(* Logix 5000 project; controller Drives_Line1 1756-L72 rev 20.13; software revision 20.04; part 11 of 21 *)
(* tags used below, declared in another part *)
   Bridle_02_FB_Count_Old : DINT;
   Bridle_02_Max_FBcounts : REAL;
   Bridle_02_SpdTrimMPS : REAL;
   Bridle_02_SpdTrimPct : REAL;
   Bridle_02a_RPMPerMPS : REAL;
   Bridle_02b_RPMPerMPS : REAL;
   IO_State_Bridle_02a : INT;
   IO_State_Bridle_02b : INT;
   IO_State_Tmp_Bridle_02a : INT;
   IO_State_Tmp_Bridle_02b : INT;
   Ons : DINT;
   PulsReset_PID : TIMER;
   TimeOn_PIDOn : TIMER;
   TofReset : TIMER;
   TonNoResponse : TIMER[3];
   TonRefOn : TIMER;
   zBridle_02_Ki_SpdTrim : REAL;
   zBridle_02_Kp_SpdTrim : REAL;
   zBridle_02_Max_rev : DINT;
   zBridle_02_MaxAccDec : REAL;
   zBridle_02_MaxTrimSpdTrim : REAL;
   zBridle_02_MinTrimSpdTrim : REAL;
   zBridle_02b_EncRes : DINT;
   Bridle_02 : UDT_Bridle_2M;
   Bridle_02_FB_Diff : DINT;
   Bridle_02_FB_Update_Valid : BOOL;
   Bridle_02_Rev_mm : REAL;
   Bridle_02b_FBCounts_mm : DINT;
   EntryCtrl : UDT_Control_Zone;
   In_Commands : UDT_Commands;
   In_Config : UDT_Config;
   LineCmd : UDT_Commands_Line;
   LineCtrl : UDT_Control_Line;
   LineFdbks : UDT_Feedbacks_Line;
   TaskInterval_ms : DINT;
   zConfigFromMaster : BOOL;
   zPi : REAL;
   zSimulation : BOOL;
(* P15_Bridle_02, continued *)

ROUTINE R01_From_Master   (* ladder *)
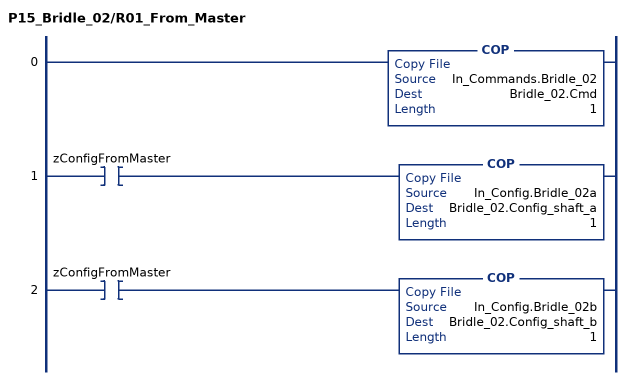
   0: COP(In_Commands.Bridle_02,Bridle_02.Cmd,1);
   1: XIC(zConfigFromMaster)COP(In_Config.Bridle_02a,Bridle_02.Config_shaft_a,1);
   2: XIC(zConfigFromMaster)COP(In_Config.Bridle_02b,Bridle_02.Config_shaft_b,1);
END_ROUTINE

ROUTINE R02_From_Drive   (* ladder *)
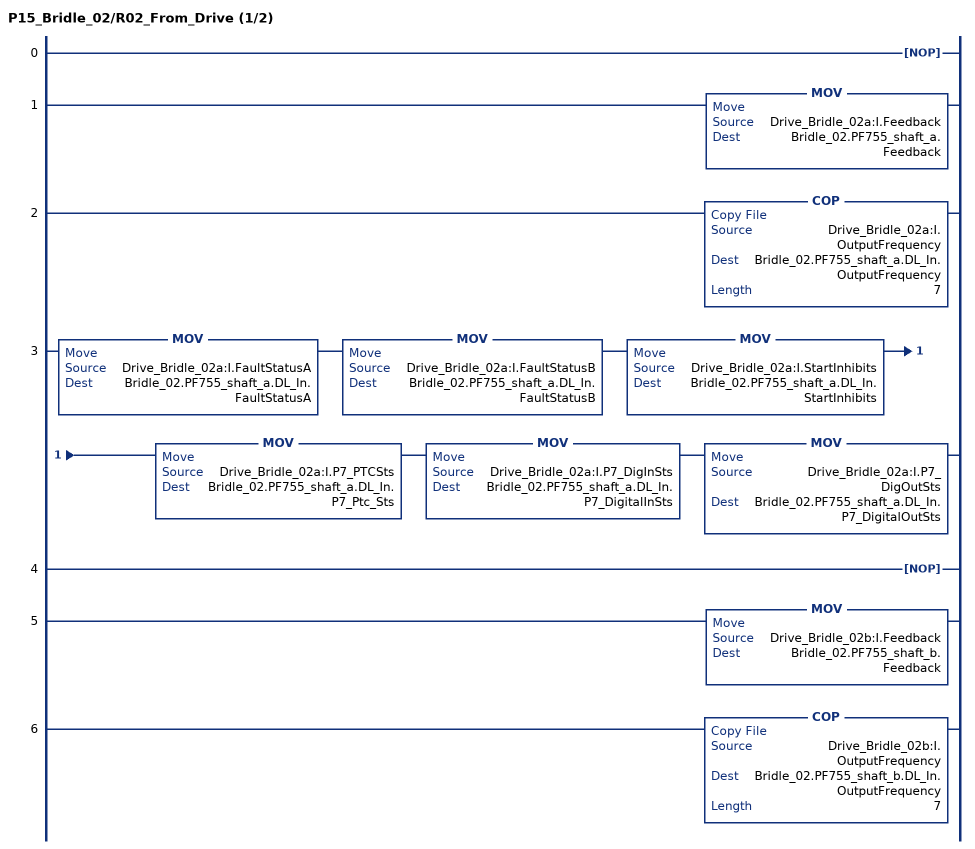
   0: NOP();
   1: MOV(Drive_Bridle_02a:I.Feedback,Bridle_02.PF755_shaft_a.Feedback);
   2: COP(Drive_Bridle_02a:I.OutputFrequency,Bridle_02.PF755_shaft_a.DL_In.OutputFrequency,7);
   3: MOV(Drive_Bridle_02a:I.FaultStatusA,Bridle_02.PF755_shaft_a.DL_In.FaultStatusA)MOV(Drive_Bridle_02a:I.FaultStatusB,Bridle_02.PF755_shaft_a.DL_In.FaultStatusB)MOV(Drive_Bridle_02a:I.StartInhibits,Bridle_02.PF755_shaft_a.DL_In.StartInhibits)MOV(Drive_Bridle_02a:I.P7_PTCSts,Bridle_02.PF755_shaft_a.DL_In.P7_Ptc_Sts)MOV(Drive_Bridle_02a:I.P7_DigInSts,Bridle_02.PF755_shaft_a.DL_In.P7_DigitalInSts)MOV(Drive_Bridle_02a:I.P7_DigOutSts,Bridle_02.PF755_shaft_a.DL_In.P7_DigitalOutSts);
   4: NOP();
   5: MOV(Drive_Bridle_02b:I.Feedback,Bridle_02.PF755_shaft_b.Feedback);
   6: COP(Drive_Bridle_02b:I.OutputFrequency,Bridle_02.PF755_shaft_b.DL_In.OutputFrequency,7);
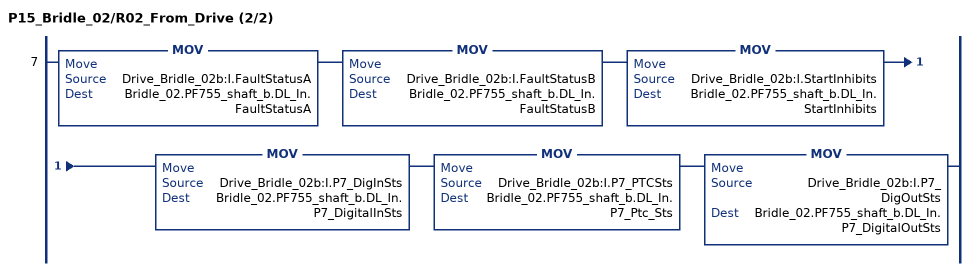
   7: MOV(Drive_Bridle_02b:I.FaultStatusA,Bridle_02.PF755_shaft_b.DL_In.FaultStatusA)MOV(Drive_Bridle_02b:I.FaultStatusB,Bridle_02.PF755_shaft_b.DL_In.FaultStatusB)MOV(Drive_Bridle_02b:I.StartInhibits,Bridle_02.PF755_shaft_b.DL_In.StartInhibits)MOV(Drive_Bridle_02b:I.P7_DigInSts,Bridle_02.PF755_shaft_b.DL_In.P7_DigitalInSts)MOV(Drive_Bridle_02b:I.P7_PTCSts,Bridle_02.PF755_shaft_b.DL_In.P7_Ptc_Sts)MOV(Drive_Bridle_02b:I.P7_DigOutSts,Bridle_02.PF755_shaft_b.DL_In.P7_DigitalOutSts);
END_ROUTINE

ROUTINE R03_Drive_Interface   (* ladder *)
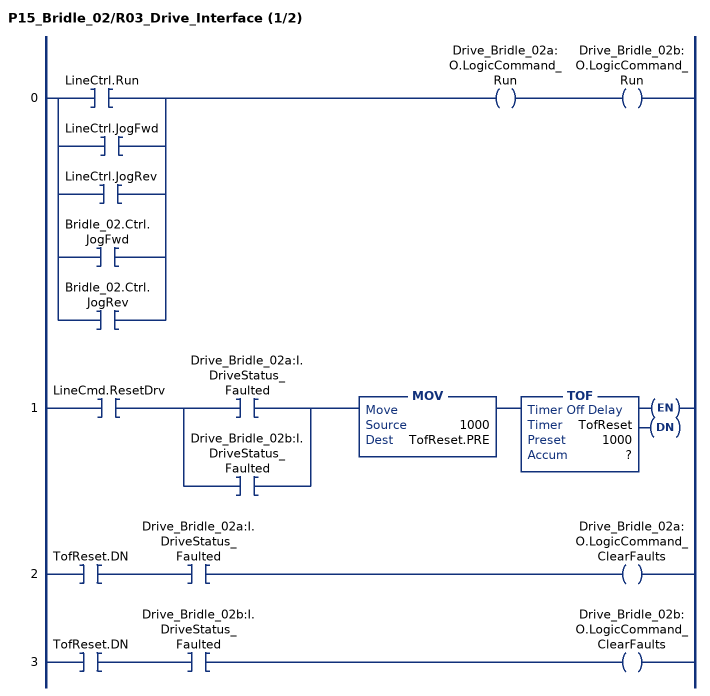
   0: [XIC(LineCtrl.Run) ,XIC(LineCtrl.JogFwd) ,XIC(LineCtrl.JogRev) ,XIC(Bridle_02.Ctrl.JogFwd) ,XIC(Bridle_02.Ctrl.JogRev) ]OTE(Drive_Bridle_02a:O.LogicCommand_Run)OTE(Drive_Bridle_02b:O.LogicCommand_Run);
   1: XIC(LineCmd.ResetDrv)[XIC(Drive_Bridle_02a:I.DriveStatus_Faulted) ,XIC(Drive_Bridle_02b:I.DriveStatus_Faulted) ]MOV(1000,TofReset.PRE)TOF(TofReset,?,?);
   2: XIC(TofReset.DN)XIC(Drive_Bridle_02a:I.DriveStatus_Faulted)OTE(Drive_Bridle_02a:O.LogicCommand_ClearFaults);
   3: XIC(TofReset.DN)XIC(Drive_Bridle_02b:I.DriveStatus_Faulted)OTE(Drive_Bridle_02b:O.LogicCommand_ClearFaults);
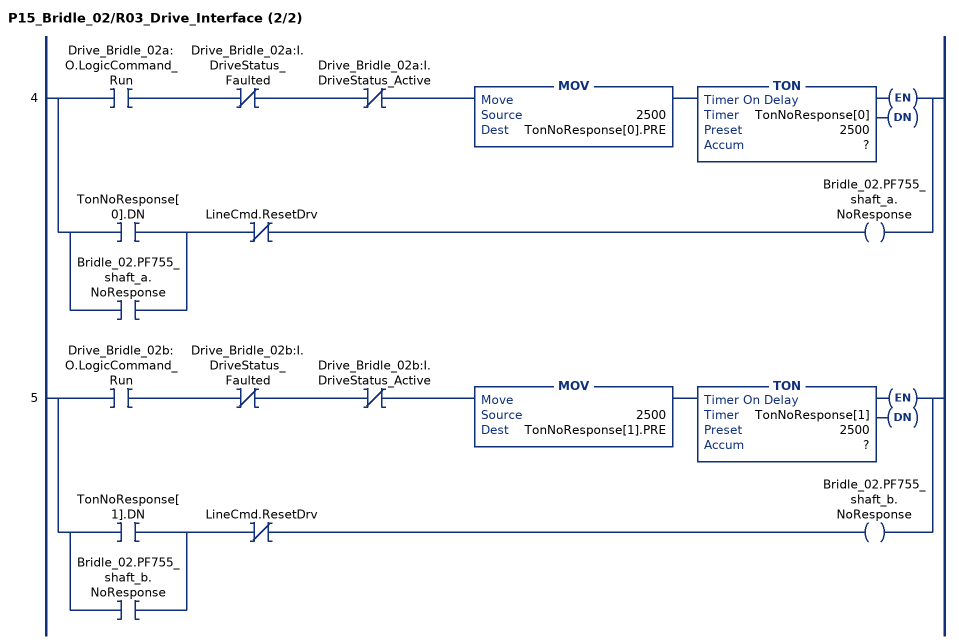
   4: [XIC(Drive_Bridle_02a:O.LogicCommand_Run) XIO(Drive_Bridle_02a:I.DriveStatus_Faulted) XIO(Drive_Bridle_02a:I.DriveStatus_Active) MOV(2500,TonNoResponse[0].PRE) TON(TonNoResponse[0],?,?) ,[XIC(TonNoResponse[0].DN) ,XIC(Bridle_02.PF755_shaft_a.NoResponse) ] XIO(LineCmd.ResetDrv) OTE(Bridle_02.PF755_shaft_a.NoResponse) ];
   5: [XIC(Drive_Bridle_02b:O.LogicCommand_Run) XIO(Drive_Bridle_02b:I.DriveStatus_Faulted) XIO(Drive_Bridle_02b:I.DriveStatus_Active) MOV(2500,TonNoResponse[1].PRE) TON(TonNoResponse[1],?,?) ,[XIC(TonNoResponse[1].DN) ,XIC(Bridle_02.PF755_shaft_b.NoResponse) ] XIO(LineCmd.ResetDrv) OTE(Bridle_02.PF755_shaft_b.NoResponse) ];
END_ROUTINE

ROUTINE R04_State   (* ladder *)
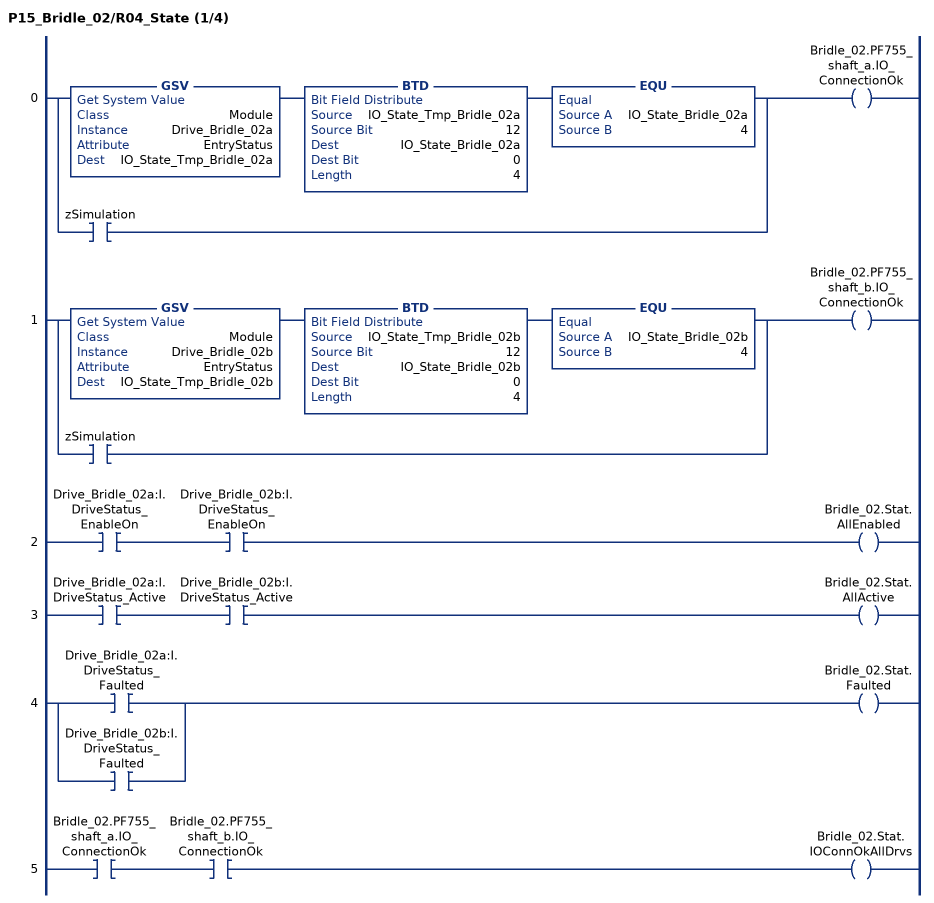
   0: [GSV(Module,Drive_Bridle_02a,EntryStatus,IO_State_Tmp_Bridle_02a) BTD(IO_State_Tmp_Bridle_02a,12,IO_State_Bridle_02a,0,4) EQU(IO_State_Bridle_02a,4) ,XIC(zSimulation) ]OTE(Bridle_02.PF755_shaft_a.IO_ConnectionOk);
   1: [GSV(Module,Drive_Bridle_02b,EntryStatus,IO_State_Tmp_Bridle_02b) BTD(IO_State_Tmp_Bridle_02b,12,IO_State_Bridle_02b,0,4) EQU(IO_State_Bridle_02b,4) ,XIC(zSimulation) ]OTE(Bridle_02.PF755_shaft_b.IO_ConnectionOk);
   2: XIC(Drive_Bridle_02a:I.DriveStatus_EnableOn)XIC(Drive_Bridle_02b:I.DriveStatus_EnableOn)OTE(Bridle_02.Stat.AllEnabled);
   3: XIC(Drive_Bridle_02a:I.DriveStatus_Active)XIC(Drive_Bridle_02b:I.DriveStatus_Active)OTE(Bridle_02.Stat.AllActive);
   4: [XIC(Drive_Bridle_02a:I.DriveStatus_Faulted) ,XIC(Drive_Bridle_02b:I.DriveStatus_Faulted) ]OTE(Bridle_02.Stat.Faulted);
   5: XIC(Bridle_02.PF755_shaft_a.IO_ConnectionOk)XIC(Bridle_02.PF755_shaft_b.IO_ConnectionOk)OTE(Bridle_02.Stat.IOConnOkAllDrvs);
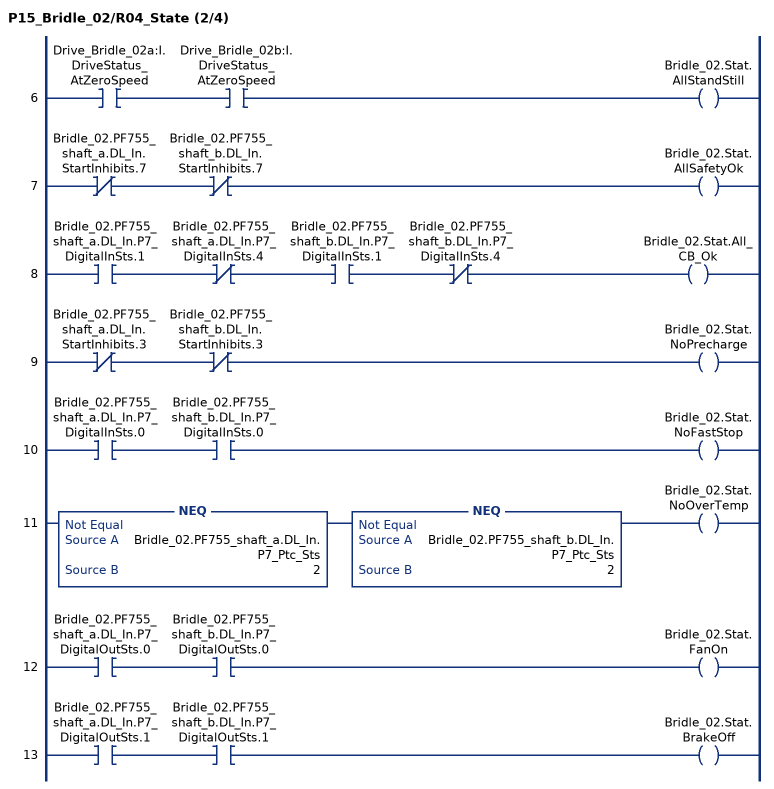
   6: XIC(Drive_Bridle_02a:I.DriveStatus_AtZeroSpeed)XIC(Drive_Bridle_02b:I.DriveStatus_AtZeroSpeed)OTE(Bridle_02.Stat.AllStandStill);
   7: XIO(Bridle_02.PF755_shaft_a.DL_In.StartInhibits.7)XIO(Bridle_02.PF755_shaft_b.DL_In.StartInhibits.7)OTE(Bridle_02.Stat.AllSafetyOk);
   8: XIC(Bridle_02.PF755_shaft_a.DL_In.P7_DigitalInSts.1)XIO(Bridle_02.PF755_shaft_a.DL_In.P7_DigitalInSts.4)XIC(Bridle_02.PF755_shaft_b.DL_In.P7_DigitalInSts.1)XIO(Bridle_02.PF755_shaft_b.DL_In.P7_DigitalInSts.4)OTE(Bridle_02.Stat.All_CB_Ok);
   9: XIO(Bridle_02.PF755_shaft_a.DL_In.StartInhibits.3)XIO(Bridle_02.PF755_shaft_b.DL_In.StartInhibits.3)OTE(Bridle_02.Stat.NoPrecharge);
   10: XIC(Bridle_02.PF755_shaft_a.DL_In.P7_DigitalInSts.0)XIC(Bridle_02.PF755_shaft_b.DL_In.P7_DigitalInSts.0)OTE(Bridle_02.Stat.NoFastStop);
   11: NEQ(Bridle_02.PF755_shaft_a.DL_In.P7_Ptc_Sts,2)NEQ(Bridle_02.PF755_shaft_b.DL_In.P7_Ptc_Sts,2)OTE(Bridle_02.Stat.NoOverTemp);
   12: XIC(Bridle_02.PF755_shaft_a.DL_In.P7_DigitalOutSts.0)XIC(Bridle_02.PF755_shaft_b.DL_In.P7_DigitalOutSts.0)OTE(Bridle_02.Stat.FanOn);
   13: XIC(Bridle_02.PF755_shaft_a.DL_In.P7_DigitalOutSts.1)XIC(Bridle_02.PF755_shaft_b.DL_In.P7_DigitalOutSts.1)OTE(Bridle_02.Stat.BrakeOff);
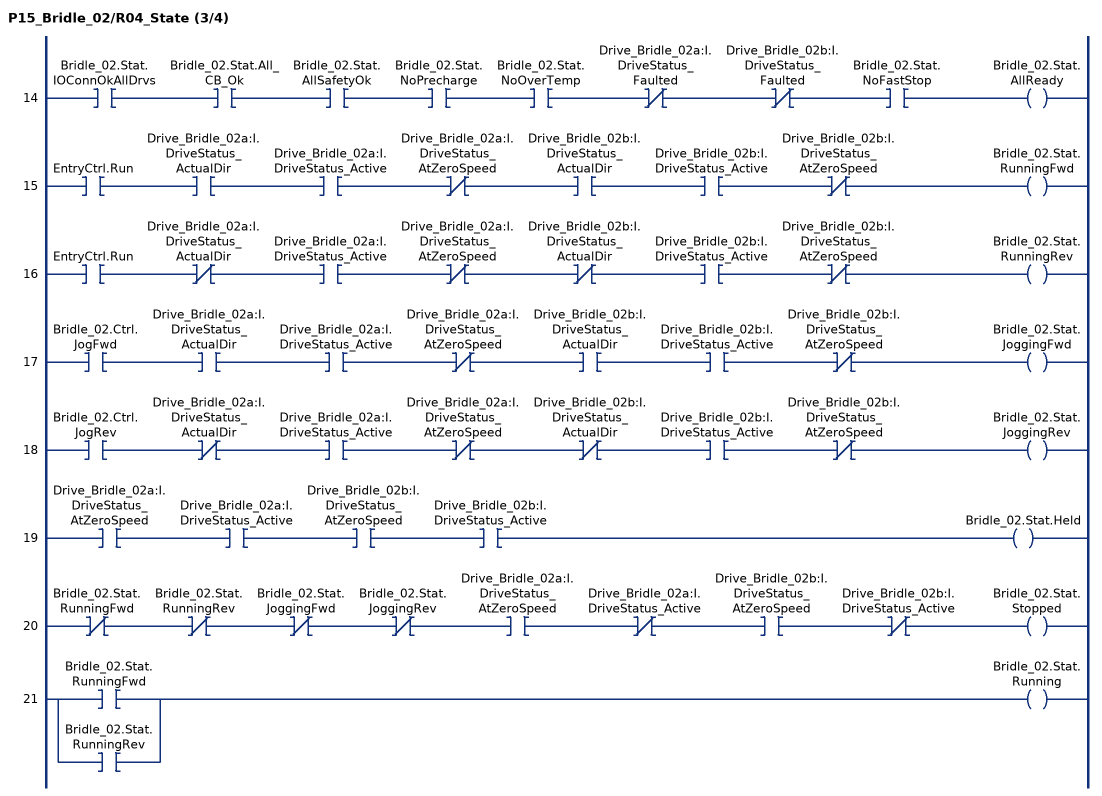
   14: XIC(Bridle_02.Stat.IOConnOkAllDrvs)XIC(Bridle_02.Stat.All_CB_Ok)XIC(Bridle_02.Stat.AllSafetyOk)XIC(Bridle_02.Stat.NoPrecharge)XIC(Bridle_02.Stat.NoOverTemp)XIO(Drive_Bridle_02a:I.DriveStatus_Faulted)XIO(Drive_Bridle_02b:I.DriveStatus_Faulted)XIC(Bridle_02.Stat.NoFastStop)OTE(Bridle_02.Stat.AllReady);
   15: XIC(EntryCtrl.Run)XIC(Drive_Bridle_02a:I.DriveStatus_ActualDir)XIC(Drive_Bridle_02a:I.DriveStatus_Active)XIO(Drive_Bridle_02a:I.DriveStatus_AtZeroSpeed)XIC(Drive_Bridle_02b:I.DriveStatus_ActualDir)XIC(Drive_Bridle_02b:I.DriveStatus_Active)XIO(Drive_Bridle_02b:I.DriveStatus_AtZeroSpeed)OTE(Bridle_02.Stat.RunningFwd);
   16: XIC(EntryCtrl.Run)XIO(Drive_Bridle_02a:I.DriveStatus_ActualDir)XIC(Drive_Bridle_02a:I.DriveStatus_Active)XIO(Drive_Bridle_02a:I.DriveStatus_AtZeroSpeed)XIO(Drive_Bridle_02b:I.DriveStatus_ActualDir)XIC(Drive_Bridle_02b:I.DriveStatus_Active)XIO(Drive_Bridle_02b:I.DriveStatus_AtZeroSpeed)OTE(Bridle_02.Stat.RunningRev);
   17: XIC(Bridle_02.Ctrl.JogFwd)XIC(Drive_Bridle_02a:I.DriveStatus_ActualDir)XIC(Drive_Bridle_02a:I.DriveStatus_Active)XIO(Drive_Bridle_02a:I.DriveStatus_AtZeroSpeed)XIC(Drive_Bridle_02b:I.DriveStatus_ActualDir)XIC(Drive_Bridle_02b:I.DriveStatus_Active)XIO(Drive_Bridle_02b:I.DriveStatus_AtZeroSpeed)OTE(Bridle_02.Stat.JoggingFwd);
   18: XIC(Bridle_02.Ctrl.JogRev)XIO(Drive_Bridle_02a:I.DriveStatus_ActualDir)XIC(Drive_Bridle_02a:I.DriveStatus_Active)XIO(Drive_Bridle_02a:I.DriveStatus_AtZeroSpeed)XIO(Drive_Bridle_02b:I.DriveStatus_ActualDir)XIC(Drive_Bridle_02b:I.DriveStatus_Active)XIO(Drive_Bridle_02b:I.DriveStatus_AtZeroSpeed)OTE(Bridle_02.Stat.JoggingRev);
   19: XIC(Drive_Bridle_02a:I.DriveStatus_AtZeroSpeed)XIC(Drive_Bridle_02a:I.DriveStatus_Active)XIC(Drive_Bridle_02b:I.DriveStatus_AtZeroSpeed)XIC(Drive_Bridle_02b:I.DriveStatus_Active)OTE(Bridle_02.Stat.Held);
   20: XIO(Bridle_02.Stat.RunningFwd)XIO(Bridle_02.Stat.RunningRev)XIO(Bridle_02.Stat.JoggingFwd)XIO(Bridle_02.Stat.JoggingRev)XIC(Drive_Bridle_02a:I.DriveStatus_AtZeroSpeed)XIO(Drive_Bridle_02a:I.DriveStatus_Active)XIC(Drive_Bridle_02b:I.DriveStatus_AtZeroSpeed)XIO(Drive_Bridle_02b:I.DriveStatus_Active)OTE(Bridle_02.Stat.Stopped);
   21: [XIC(Bridle_02.Stat.RunningFwd) ,XIC(Bridle_02.Stat.RunningRev) ]OTE(Bridle_02.Stat.Running);
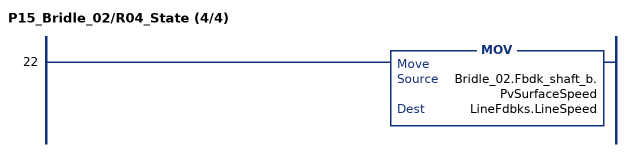
   22: MOV(Bridle_02.Fbdk_shaft_b.PvSurfaceSpeed,LineFdbks.LineSpeed);
END_ROUTINE

ROUTINE R05_Control   (* ladder *)
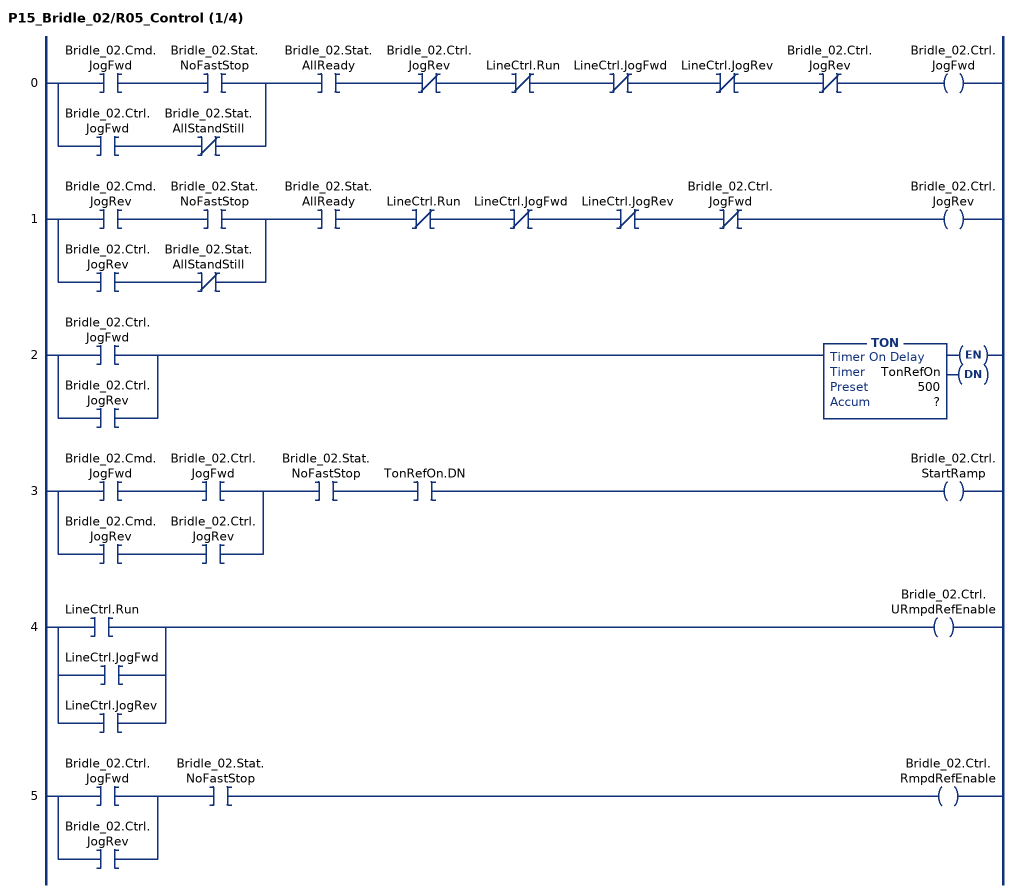
   0: [XIC(Bridle_02.Cmd.JogFwd) XIC(Bridle_02.Stat.NoFastStop) ,XIC(Bridle_02.Ctrl.JogFwd) XIO(Bridle_02.Stat.AllStandStill) ]XIC(Bridle_02.Stat.AllReady)XIO(Bridle_02.Ctrl.JogRev)XIO(LineCtrl.Run)XIO(LineCtrl.JogFwd)XIO(LineCtrl.JogRev)XIO(Bridle_02.Ctrl.JogRev)OTE(Bridle_02.Ctrl.JogFwd);
   1: [XIC(Bridle_02.Cmd.JogRev) XIC(Bridle_02.Stat.NoFastStop) ,XIC(Bridle_02.Ctrl.JogRev) XIO(Bridle_02.Stat.AllStandStill) ]XIC(Bridle_02.Stat.AllReady)XIO(LineCtrl.Run)XIO(LineCtrl.JogFwd)XIO(LineCtrl.JogRev)XIO(Bridle_02.Ctrl.JogFwd)OTE(Bridle_02.Ctrl.JogRev);
   2: [XIC(Bridle_02.Ctrl.JogFwd) ,XIC(Bridle_02.Ctrl.JogRev) ]TON(TonRefOn,?,?);
   3: [XIC(Bridle_02.Cmd.JogFwd) XIC(Bridle_02.Ctrl.JogFwd) ,XIC(Bridle_02.Cmd.JogRev) XIC(Bridle_02.Ctrl.JogRev) ]XIC(Bridle_02.Stat.NoFastStop)XIC(TonRefOn.DN)OTE(Bridle_02.Ctrl.StartRamp);
   4: [XIC(LineCtrl.Run) ,XIC(LineCtrl.JogFwd) ,XIC(LineCtrl.JogRev) ]OTE(Bridle_02.Ctrl.URmpdRefEnable);
   5: [XIC(Bridle_02.Ctrl.JogFwd) ,XIC(Bridle_02.Ctrl.JogRev) ]XIC(Bridle_02.Stat.NoFastStop)OTE(Bridle_02.Ctrl.RmpdRefEnable);
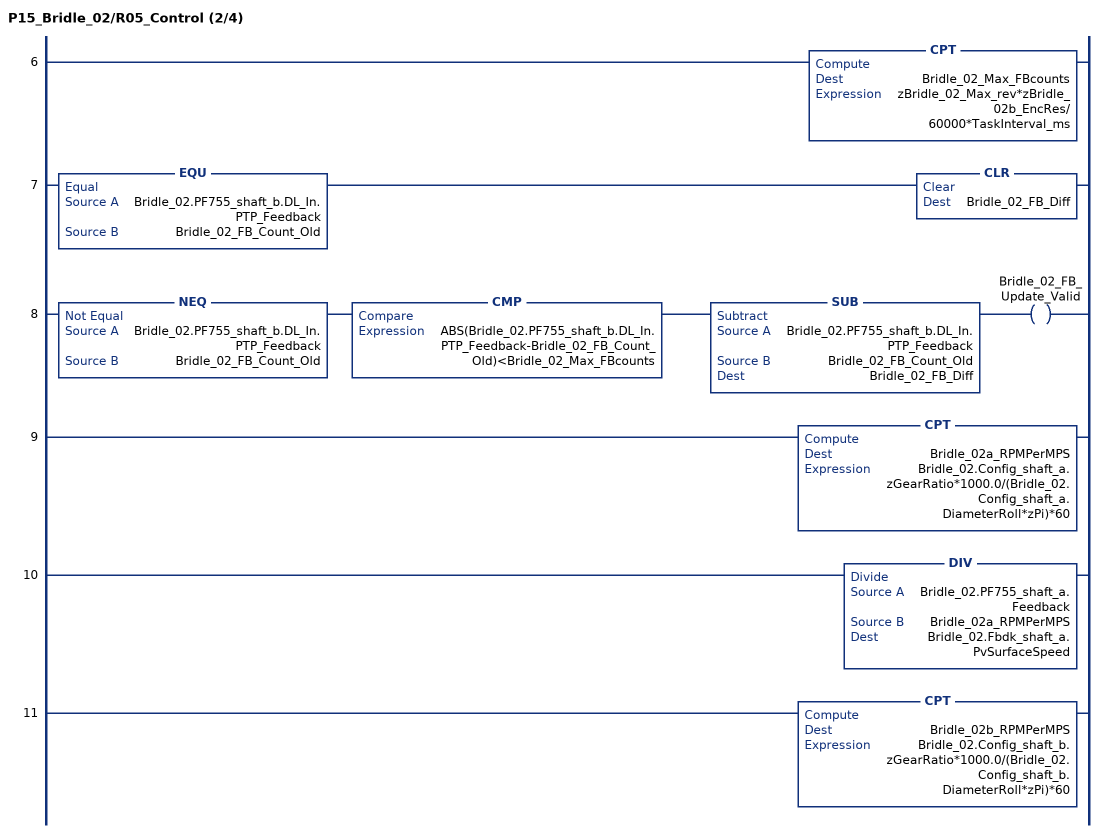
   6: CPT(Bridle_02_Max_FBcounts,zBridle_02_Max_rev*zBridle_02b_EncRes/60000*TaskInterval_ms);
   7: EQU(Bridle_02.PF755_shaft_b.DL_In.PTP_Feedback,Bridle_02_FB_Count_Old)CLR(Bridle_02_FB_Diff);
   8: NEQ(Bridle_02.PF755_shaft_b.DL_In.PTP_Feedback,Bridle_02_FB_Count_Old)CMP(ABS(Bridle_02.PF755_shaft_b.DL_In.PTP_Feedback-Bridle_02_FB_Count_Old)<Bridle_02_Max_FBcounts)SUB(Bridle_02.PF755_shaft_b.DL_In.PTP_Feedback,Bridle_02_FB_Count_Old,Bridle_02_FB_Diff)OTE(Bridle_02_FB_Update_Valid);
   9: CPT(Bridle_02a_RPMPerMPS,Bridle_02.Config_shaft_a.zGearRatio*1000.0/(Bridle_02.Config_shaft_a.DiameterRoll*zPi)*60);
   10: DIV(Bridle_02.PF755_shaft_a.Feedback,Bridle_02a_RPMPerMPS,Bridle_02.Fbdk_shaft_a.PvSurfaceSpeed);
   11: CPT(Bridle_02b_RPMPerMPS,Bridle_02.Config_shaft_b.zGearRatio*1000.0/(Bridle_02.Config_shaft_b.DiameterRoll*zPi)*60);
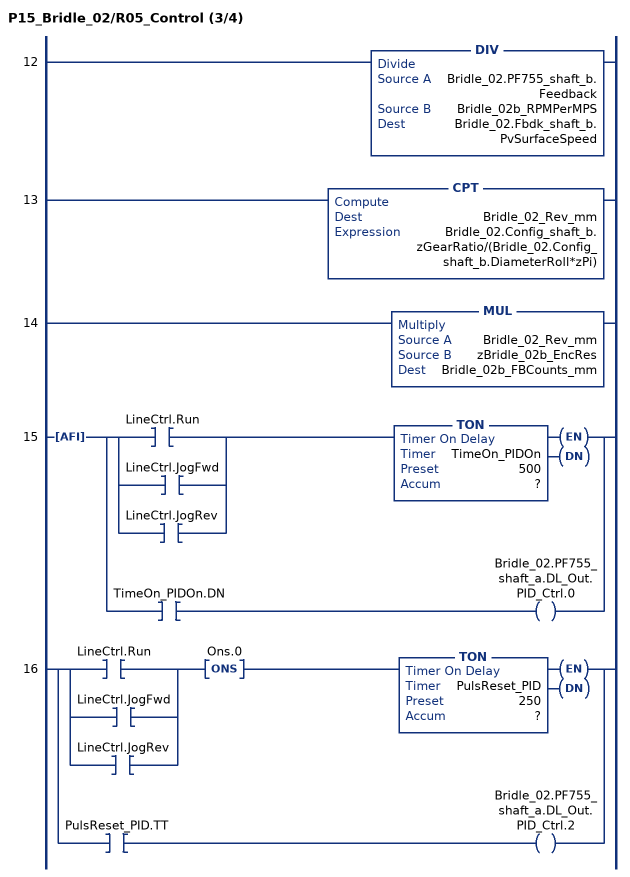
   12: DIV(Bridle_02.PF755_shaft_b.Feedback,Bridle_02b_RPMPerMPS,Bridle_02.Fbdk_shaft_b.PvSurfaceSpeed);
   13: CPT(Bridle_02_Rev_mm,Bridle_02.Config_shaft_b.zGearRatio/(Bridle_02.Config_shaft_b.DiameterRoll*zPi));
   14: MUL(Bridle_02_Rev_mm,zBridle_02b_EncRes,Bridle_02b_FBCounts_mm);
   15: AFI()[[XIC(LineCtrl.Run) ,XIC(LineCtrl.JogFwd) ,XIC(LineCtrl.JogRev) ] TON(TimeOn_PIDOn,?,?) ,XIC(TimeOn_PIDOn.DN) OTE(Bridle_02.PF755_shaft_a.DL_Out.PID_Ctrl.0) ];
   16: [[XIC(LineCtrl.Run) ,XIC(LineCtrl.JogFwd) ,XIC(LineCtrl.JogRev) ] ONS(Ons.0) TON(PulsReset_PID,?,?) ,XIC(PulsReset_PID.TT) OTE(Bridle_02.PF755_shaft_a.DL_Out.PID_Ctrl.2) ];
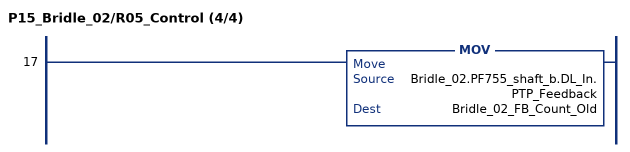
   17: MOV(Bridle_02.PF755_shaft_b.DL_In.PTP_Feedback,Bridle_02_FB_Count_Old);
END_ROUTINE

ROUTINE R11_LoadSharing   (* function block diagram *)
   SHEET 1   // Load sharing speed trim percentage
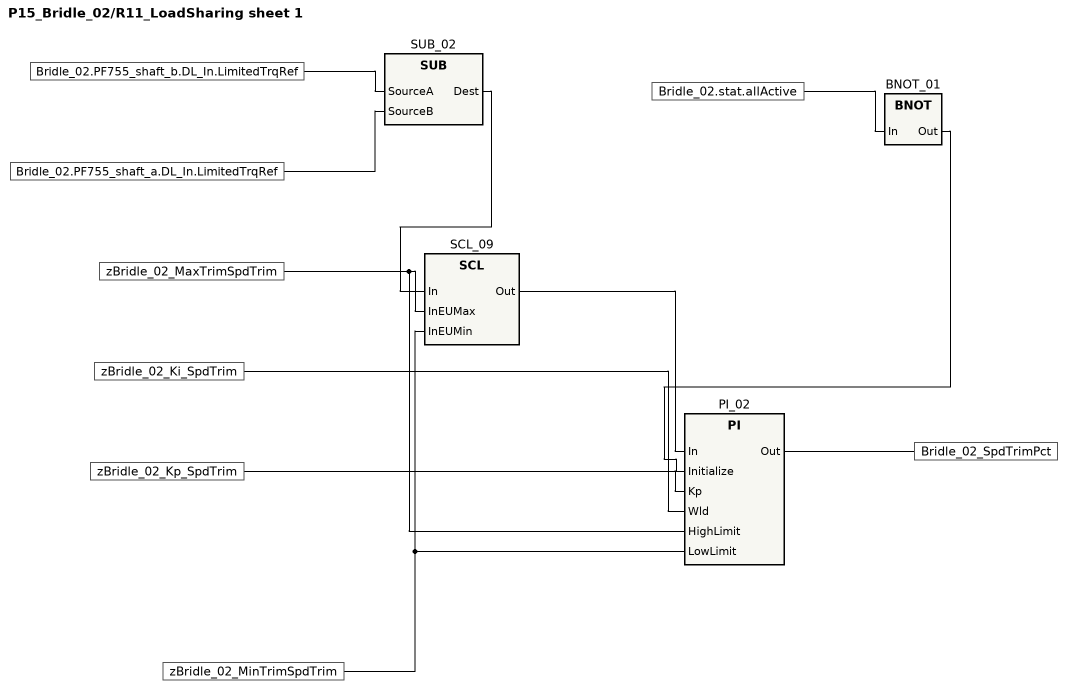
   SUB_02 : SUB(SourceA := Bridle_02.PF755_shaft_b.DL_In.LimitedTrqRef, SourceB := Bridle_02.PF755_shaft_a.DL_In.LimitedTrqRef);
   SCL_09 : SCL(In := SUB_02.Dest, InEUMax := zBridle_02_MaxTrimSpdTrim, InEUMin := zBridle_02_MinTrimSpdTrim);
   BNOT_01 : BNOT(In := Bridle_02.stat.allActive);
   PI_02 : PI(In := SCL_09.Out, Initialize := BNOT_01.Out, Kp := zBridle_02_Kp_SpdTrim, Wld := zBridle_02_Ki_SpdTrim, HighLimit := zBridle_02_MaxTrimSpdTrim, LowLimit := zBridle_02_MinTrimSpdTrim);
   Bridle_02_SpdTrimPct := PI_02.Out;
   SHEET 2   // Calculate speed trim mps
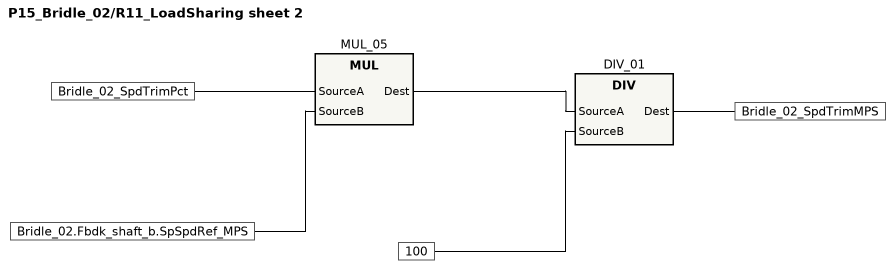
   MUL_05 : MUL(SourceA := Bridle_02_SpdTrimPct, SourceB := Bridle_02.Fbdk_shaft_b.SpSpdRef_MPS);
   DIV_01 : DIV(SourceA := MUL_05.Dest, SourceB := 100);
   Bridle_02_SpdTrimMPS := DIV_01.Dest;
END_ROUTINE

ROUTINE R12_DriveRef   (* function block diagram *)
   SHEET 1   // Select jog speed reference
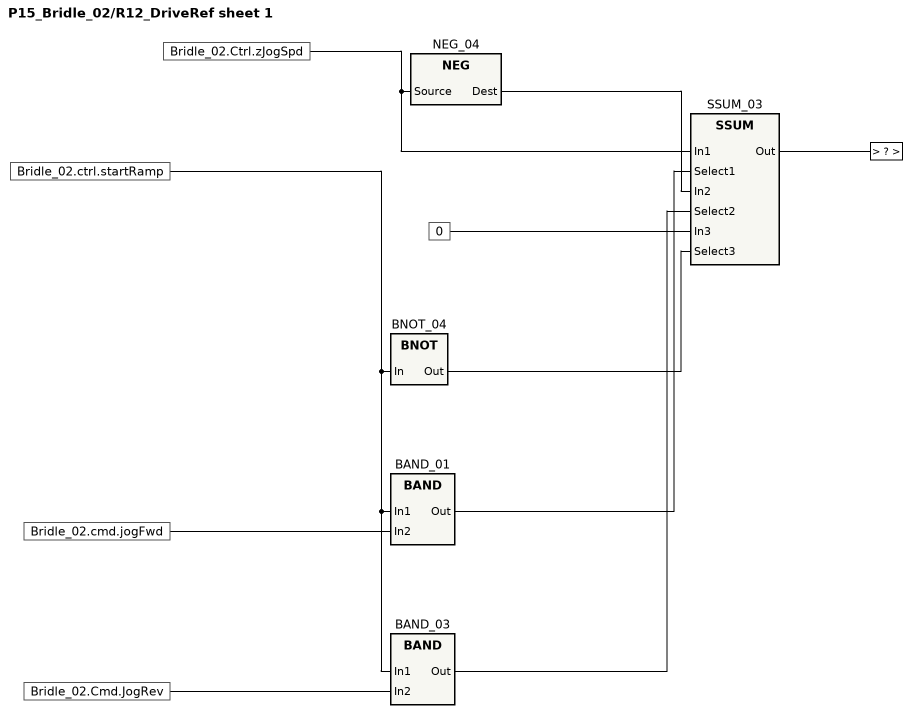
   BNOT_04 : BNOT(In := Bridle_02.ctrl.startRamp);
   BAND_01 : BAND(In1 := Bridle_02.ctrl.startRamp, In2 := Bridle_02.cmd.jogFwd);
   BAND_03 : BAND(In1 := Bridle_02.ctrl.startRamp, In2 := Bridle_02.Cmd.JogRev);
   NEG_04 : NEG(Source := Bridle_02.Ctrl.zJogSpd);
   SSUM_03 : SSUM(In1 := Bridle_02.Ctrl.zJogSpd, Select1 := BAND_01.Out, In2 := NEG_04.Dest, Select2 := BAND_03.Out, In3 := 0, Select3 := BNOT_04.Out);
   WIRE(?) := SSUM_03.Out;
   SHEET 2   // S-Curve
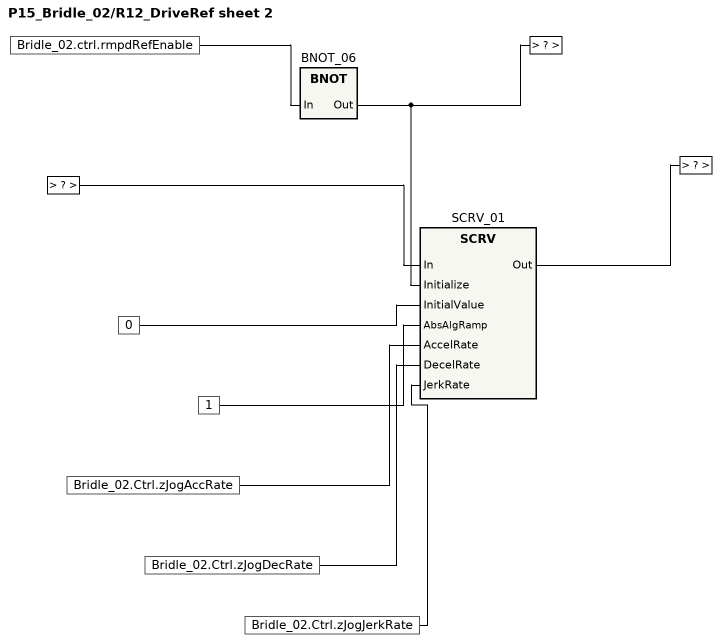
   BNOT_06 : BNOT(In := Bridle_02.ctrl.rmpdRefEnable);
   WIRE(?) := BNOT_06.Out;
   SCRV_01 : SCRV(In := WIRE(?), Initialize := BNOT_06.Out, InitialValue := 0, AbsAlgRamp := 1, AccelRate := Bridle_02.Ctrl.zJogAccRate, DecelRate := Bridle_02.Ctrl.zJogDecRate, JerkRate := Bridle_02.Ctrl.zJogJerkRate);
   WIRE(?) := SCRV_01.Out;
   SHEET 3   // Select ramped/unramped reference
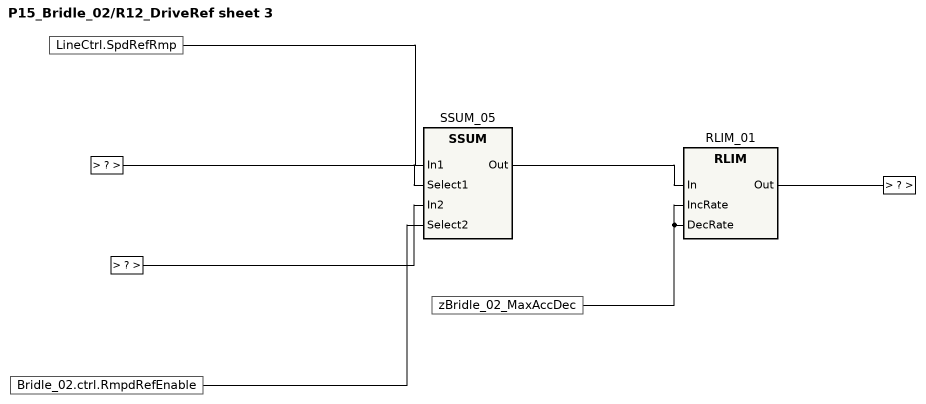
   SSUM_05 : SSUM(In1 := LineCtrl.SpdRefRmp, Select1 := WIRE(?), In2 := WIRE(?), Select2 := Bridle_02.ctrl.RmpdRefEnable);
   RLIM_01 : RLIM(In := SSUM_05.Out, IncRate := zBridle_02_MaxAccDec, DecRate := zBridle_02_MaxAccDec);
   WIRE(?) := RLIM_01.Out;
   SHEET 4   // Final speed reference
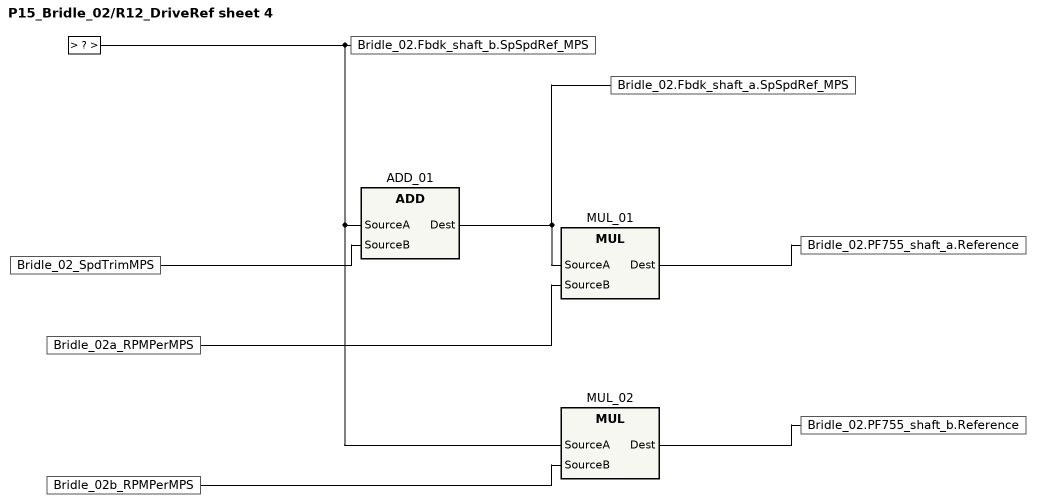
   Bridle_02.Fbdk_shaft_b.SpSpdRef_MPS := WIRE(?);
   ADD_01 : ADD(SourceA := WIRE(?), SourceB := Bridle_02_SpdTrimMPS);
   MUL_01 : MUL(SourceA := ADD_01.Dest, SourceB := Bridle_02a_RPMPerMPS);
   MUL_02 : MUL(SourceA := WIRE(?), SourceB := Bridle_02b_RPMPerMPS);
   Bridle_02.Fbdk_shaft_a.SpSpdRef_MPS := ADD_01.Dest;
   Bridle_02.PF755_shaft_a.Reference := MUL_01.Dest;
   Bridle_02.PF755_shaft_b.Reference := MUL_02.Dest;
END_ROUTINE
